(* IEC 61131-3 sources: myCodes/Stone/07.02.2022 - OOPs Approach/MPx_One_New/Mpx_One_Source_Code/MPx_One/3. USHPXMPX010A1/USHPXMPX010A1/MPXone_Medium/Gui/Actions, 31 files *)

(* ---- ALM_HystPROGRAM_RELEASE.st ---- *)
USING System;
USING System.UI;
USING HEOneRow;

FUNCTION ALM_HystPROGRAM_RELEASE
	VAR_INPUT
		keyPressed:UINT;
		keyCounter:UINT;
	END_VAR

    currMenuLevel := 2;

    GoToLoop(LoopList#ALM_LOG);

END_FUNCTION

(* ---- ALM_menu_ESC_PROGRAM_RELEASE.st ---- *)
USING System;
USING System.UI;
USING HEOneRow;

FUNCTION ALM_menu_ESC_PROGRAM_RELEASE
	VAR_INPUT
		keyPressed:UINT;
		keyCounter:UINT;
	END_VAR

    currMenuLevel := 1;
    currMenu := 4;
    GoToMask(MaskList#ALM);

END_FUNCTION

(* ---- ALM_ParamPROGRAM_RELEASE.st ---- *)
USING System;
USING System.UI;
USING HEOneRow;

FUNCTION ALM_ParamPROGRAM_RELEASE
	VAR_INPUT
		keyPressed:UINT;
		keyCounter:UINT;
	END_VAR

    currMenuLevel := 2;
    GoToLoop(LoopList#ALM_Param);

END_FUNCTION

(* ---- checkPassword.st ---- *)
USING System;
USING System.UI;
USING HEOneRow;

FUNCTION checkPassword
	VAR_INPUT
		keyPressed:UINT;
		keyCounter:UINT;
	END_VAR

    IF tmpPassword = TO_USINT(PwdDisplay) THEN
        GoToLoop(LoopList#Menu);
        blockHmi := TRUE;

        tmpPassword := 0;

        currMenu := 1; // Vis Menu
        currMenuLevel := 0; // Menu level
    ELSE
        // Wrong password
        LedBlinkArrow := FALSE;
        WrongPsw := TRUE;
        blockHmi := TRUE;
        GoToLoop(LoopList#Main);
    END_IF;

END_FUNCTION

(* ---- CntPRG.st ---- *)
USING System;
USING System.UI;
USING HEOneRow;

FUNCTION CntPRG
	VAR_INPUT
		keyPressed:UINT;
		keyCounter:UINT;
	END_VAR

    //DispMngInst.StartSync(DownloadDir#ACUtoHMI);
    NewDispPrompt := FALSE;
    GoToLoop(LoopList#Main);

END_FUNCTION

(* ---- Dir_CleanPRG.st ---- *)
USING System;
USING System.UI;
USING HEOneRow;

FUNCTION Dir_CleanPRG
	VAR_INPUT
		keyPressed:UINT;
		keyCounter:UINT;
	END_VAR

    ManClean := NOT ManClean;
END_FUNCTION

(* ---- Dir_ContCyclPRG.st ---- *)
USING System;
USING System.UI;
USING HEOneRow;

FUNCTION Dir_ContCyclPRG
	VAR_INPUT
		keyPressed:UINT;
		keyCounter:UINT;
	END_VAR

    ManContCycle_byDisplay := NOT ManContCycle_byDisplay;

END_FUNCTION

(* ---- Dir_DefrostPRG.st ---- *)
USING System;
USING System.UI;
USING HEOneRow;

FUNCTION Dir_DefrostPRG
	VAR_INPUT
		keyPressed:UINT;
		keyCounter:UINT;
	END_VAR

    ManDfr := NOT ManDfr;

END_FUNCTION

(* ---- Dir_LightPRG.st ---- *)
USING System;
USING System.UI;
USING HEOneRow;

FUNCTION Dir_LightPRG
	VAR_INPUT
		keyPressed:UINT;
		keyCounter:UINT;
	END_VAR

    LightsOn := NOT LightsOn;
END_FUNCTION

(* ---- Dir_NetDefrostPRG.st ---- *)
USING System;
USING System.UI;
USING HEOneRow;

FUNCTION Dir_NetDefrostPRG
	VAR_INPUT
		keyPressed:UINT;
		keyCounter:UINT;
	END_VAR

    NetworkDfr := NOT NetworkDfr;

END_FUNCTION

(* ---- Dir_OnOffPRG.st ---- *)
USING System;
USING System.UI;
USING HEOneRow;

FUNCTION Dir_OnOffPRG
	VAR_INPUT
		keyPressed:UINT;
		keyCounter:UINT;
	END_VAR

    IF NOT(DigitalInputs.Fct.RemoteOff) THEN // TRAC #99: Allow to change the status from UI only if remote off is not active
        KeyboardOnOff := NOT KeyboardOnOff;
        //        UnitStatus := NOT UnitStatus;
    END_IF;

END_FUNCTION

(* ---- DisPRG.st ---- *)
USING System;
USING System.UI;
USING HEOneRow;

FUNCTION DisPRG
	VAR_INPUT
		keyPressed:UINT;
		keyCounter:UINT;
	END_VAR

    //DispMngInst.StartSync(DownloadDir#HMItoACU);
    NewDispPrompt := FALSE;
    GoToLoop(LoopList#Main);

END_FUNCTION

(* ---- doNothing.st ---- *)
USING System;
USING System.UI;
USING HEOneRow;

FUNCTION doNothing
	VAR_INPUT
		keyPressed:UINT;
		keyCounter:UINT;
	END_VAR

END_FUNCTION

(* ---- GlassGUIALARM.st ---- *)
USING System;
USING System.UI;
USING HEOneRow;

FUNCTION GlassGUIALARM
	VAR_INPUT
		keyPressed:UINT;
		keyCounter:UINT;
	END_VAR

    IF AckAlm AND keyCounter < 30 THEN
        // Block user interface
        IF NOT EnKeyboard THEN
            RETURN;
        END_IF;

        IF (NOT OrAlrm) AND (NOT OrWarning) THEN
            RETURN;
        END_IF;

        GoToMask(MaskList#ActiveAlarms);
        //InsideLoopAlrm := TRUE;
        Navigation := TRUE;
    END_IF;

    IF NOT Alarms.Al.Warn_Door.Info.Trigger THEN
        AckAlm := TRUE;
    END_IF;

END_FUNCTION

(* ---- GoToLastRTC.st ---- *)
USING System;
USING System.UI;
USING HEOneRow;

FUNCTION GoToLastRTC
	VAR_INPUT
		keyPressed:UINT;
		keyCounter:UINT;
	END_VAR

    //GoToMask(MaskList#tc);
END_FUNCTION

(* ---- GoToMain.st ---- *)
USING System;
USING System.UI;
USING HEOneRow;

FUNCTION GoToMain
	VAR_INPUT
		keyPressed:UINT;
		keyCounter:UINT;
	END_VAR

    // Turn off LEDS used for menu
    LedOnArrow := FALSE;
    LedBlinkArrow := FALSE;

    /*rkLed[0] := FALSE;
    rkLed[1] := FALSE;
    rkLed[2] := FALSE;
    rkLed[3] := FALSE;
    lkLed[0] := FALSE;
    lkLed[1] := FALSE;
    lkLed[2] := FALSE;
    lkLed[3] := FALSE;
    lkLed[4] := FALSE;
    LedAlarm := FALSE;*/

    Navigation := FALSE;
    InsideLoopDirFunct := FALSE;
    currMenuLevel := 0;

    blockHmi := TRUE;
    BasicVisualiz := FALSE;

    GoToMask(MaskList#mMain);
END_FUNCTION

(* ---- GoToPassword.st ---- *)
USING System;
USING System.UI;
USING HEOneRow;

FUNCTION GoToPassword
	VAR_INPUT
		keyPressed:UINT;
		keyCounter:UINT;
	END_VAR

    // Block user interface
    IF NOT EnKeyboard THEN
        RETURN;
    END_IF;

    IF keyCounter>30 AND BlockHmi = FALSE THEN
        blockHmi := TRUE;
        Navigation := TRUE;
        GoToMask(MaskList#mPassword);
    END_IF;

END_FUNCTION

(* ---- HSx_PROGRAM_RELEASE.st ---- *)
USING System;
USING System.UI;
USING HEOneRow;

FUNCTION HSx_PROGRAM_RELEASE
	VAR_INPUT
		keyPressed:UINT;
		keyCounter:UINT;
	END_VAR

    CASE GetCurrentMask() OF
        TO_UINT(MaskList#HS0) : IdxVis_AlrmHyst := 1;
        TO_UINT(MaskList#HS1) : IdxVis_AlrmHyst := 2;
        TO_UINT(MaskList#HS2) : IdxVis_AlrmHyst := 3;
        TO_UINT(MaskList#HS3) : IdxVis_AlrmHyst := 4;
        TO_UINT(MaskList#HS4) : IdxVis_AlrmHyst := 5;
        TO_UINT(MaskList#HS5) : IdxVis_AlrmHyst := 6;
        TO_UINT(MaskList#HS6) : IdxVis_AlrmHyst := 7;
        TO_UINT(MaskList#HS7) : IdxVis_AlrmHyst := 8;
        TO_UINT(MaskList#HS8) : IdxVis_AlrmHyst := 9;
        TO_UINT(MaskList#HS9) : IdxVis_AlrmHyst := 10;
    END_CASE;

   GoToMask(MaskList#ShowAlrmHyst);

END_FUNCTION

(* ---- MenuPRG.st ---- *)
USING System;
USING System.UI;
USING HEOneRow;

FUNCTION MenuPRG
	VAR_INPUT
		keyPressed:UINT;
		keyCounter:UINT;
	END_VAR

    IF keyCounter >30 AND NOT blockHmi THEN
        blockHmi := TRUE;

        IF currMenuLevel = 0 THEN
            GoToMask(MaskList#mMain);

        ELSE
            CASE currMenu OF
                1: GoToMask(MaskList#VIS);
                2: GoToMask(MaskList#CTL);
                3: GoToMask(MaskList#DEF);
                4: GoToMask(MaskList#ALM);
                5: GoToMask(MaskList#FAN);
                6: GoToMask(MaskList#EVD);
                7: GoToMask(MaskList#CNF);
            ELSE
                GoToLoop(LoopList#Menu);
            END_CASE;

            currMenuLevel := 0;
        END_IF;
    END_IF;

END_FUNCTION

(* ---- MenuPROGRAM_RELEASE.st ---- *)
USING System;
USING System.UI;

NAMESPACE HEOneRow

FUNCTION MenuPROGRAM_RELEASE
	VAR_INPUT
		keyPressed:UINT;
		keyCounter:UINT;
	END_VAR

    IF keyCounter < 30 AND NOT blockHmi THEN

        IF BasicVisualiz AND GetCurrentMask() = GetLastMaskInLoop(gui.currentLoop) THEN
            GoToMask(MaskList#mMain);
            BasicVisualiz := FALSE;
            LedOnArrow := FALSE;
            PrbVisualiz := FALSE;
            RETURN;
        END_IF;

        CASE currMenuLevel OF
            0: // At function selection

            IF isProdBasicVersion AND currMenu = 6 THEN
                currMenu := 7;
            END_IF;

            CASE currMenu OF
                1: GoToLoop(LoopList#VIS_Loop);
                2: GoToLoop(LoopList#CTL_Param);
                3: GoToLoop(LoopList#dEF_Param);
                4: GoToLoop(LoopList#ALM_menu);
                5: GoToLoop(LoopList#FAN_Param);
                {IF DEF(MPXONE_MEDIUM)}
                6: GoToLoop(LoopList#EVD_Param);
                {ENDIF}
                7: GoToLoop(LoopList#CNF_Param);
                8: GoToLoop(LoopList#rtC_Param);
            ELSE
                GoToLoop(LoopList#Menu);
            END_CASE;

            currMenuLevel := 1;

            1: // editing the value
            GoToNextField();

            // Or exiting
            IF GetCurrentMask() = GetLastMaskInLoop(gui.currentLoop) THEN
                CASE currMenu OF
                    1: GoToMask(MaskList#VIS);
                    2: GoToMask(MaskList#CTL);
                    3: GoToMask(MaskList#DEF);
                    4: GoToMask(MaskList#ALM);
                    5: GoToMask(MaskList#FAN);
                    6: GoToMask(MaskList#EVD);
                    7: GoToMask(MaskList#CNF);
                    8: GoToMask(MaskList#RtC);
                ELSE
                    GoToLoop(LoopList#Menu);
                END_CASE;

                currMenuLevel := 0;
                currMenu_SecondLev := 0;
            END_IF;

            2: // editing the value
            GoToNextField();

            // Or exiting
            IF GetCurrentMask() = GetLastMaskInLoop(gui.currentLoop) THEN
                CASE currMenu_SecondLev OF
                    0: GoToMask(MaskList#ALM_Param);
                    1: GoToMask(MaskList#ALM_Hyst);
                ELSE
                    GoToMask(MaskList#ALM);
                END_CASE;
                currMenu := 4;
                currMenuLevel := 1;
            END_IF;

        END_CASE;

    END_IF;

    blockHmi := FALSE;

END_FUNCTION

END_NAMESPACE

(* ---- MenuSecondUPDOWN.st ---- *)
USING System;
USING System.UI;
USING HEOneRow;

FUNCTION MenuSecondUPDOWN
	VAR_INPUT
		keyPressed:UINT;
		keyCounter:UINT;
	END_VAR

    // keyPressed = 14 tasto UP
    IF keyPressed = 14 THEN
        currMenu_SecondLev := currMenu_SecondLev - 1;
        IF currMenu_SecondLev > 2 THEN // CurrMenu is unsigned so it will become 255 insthead of -1
            currMenu_SecondLev := 2;
        END_IF;
        GoToPreviousMask();
    END_IF;

    // keyPressed = 15 tasto DOWN
    IF keyPressed = 15 THEN
        currMenu_SecondLev := currMenu_SecondLev + 1;
        IF currMenu_SecondLev > 2 THEN
            currMenu_SecondLev := 0;
        END_IF;
        GoToNextMask();
    END_IF;

END_FUNCTION

(* ---- MenuUPDOWN.st ---- *)
USING System;
USING System.UI;
USING HEOneRow;

FUNCTION MenuUPDOWN
	VAR_INPUT
		keyPressed:UINT;
		keyCounter:UINT;
	END_VAR

    // keyPressed = 14 tasto UP
    IF keyPressed = 14 THEN
        currMenu := currMenu - 1;
        IF currMenu > MENU_ITEMS THEN // CurrMenu is unsigned so it will become 255 insthead of -1
            currMenu := MENU_ITEMS;
        END_IF;
        GoToPreviousMask();
    END_IF;

    // keyPressed = 15 tasto DOWN
    IF keyPressed = 15 THEN
        currMenu := currMenu + 1;
        IF currMenu > MENU_ITEMS THEN
            currMenu := 0;
        END_IF;
        GoToNextMask();
    END_IF;

END_FUNCTION

(* ---- mMainALARM.st ---- *)
USING System;
USING System.UI;
USING HEOneRow;

FUNCTION mMainALARM
	VAR_INPUT
		keyPressed:UINT;
		keyCounter:UINT;
	END_VAR

//    IF AckAlm THEN
//        GoToMask(MaskList#ActiveAlarms);
//        //InsideLoopAlrm := TRUE;
//        Navigation := TRUE;
//    END_IF;

    // Block user interface
    IF NOT EnKeyboard THEN
        RETURN;
    END_IF;

    // Long press to reset alarm
    IF keyCounter>30 AND blockHmi = FALSE THEN
        AlrmRes := TRUE;
    END_IF;

END_FUNCTION

(* ---- mMainPRG.st ---- *)
USING System;
USING System.UI;
USING HEOneRow;

FUNCTION mMainPRG
	VAR_INPUT
		keyPressed:UINT;
		keyCounter:UINT;
	END_VAR

    IF keyCounter>30 AND firstCycle AND NOT blockHmi THEN
        blockHmi := TRUE;
        StartupReset := TRUE;
        GoToMask(MaskList#DefSelection);
        RETURN;
    END_IF;

    IF firstCycle THEN
        RETURN;
    END_IF;

    // Block user interface
    IF NOT EnKeyboard THEN
        RETURN;
    END_IF;

    IF keyCounter>30 AND blockHmi = FALSE THEN
        blockHmi := TRUE;
        Navigation := TRUE;
        GoToMask(MaskList#mTxtPsd);
    END_IF;

END_FUNCTION

(* ---- mMainPROGRAM_RELEASE.st ---- *)
USING System;
USING System.UI;
USING HEOneRow;

FUNCTION mMainPROGRAM_RELEASE
	VAR_INPUT
		keyPressed:UINT;
		keyCounter:UINT;
	END_VAR

    // Block user interface
    IF NOT EnKeyboard THEN
        RETURN;
    END_IF;

    Navigation := FALSE;
    InsideLoopDirFunct := FALSE;

    IF blockHmi = FALSE AND keyCounter <30 AND EnDirFunct AND NOT firstCycle THEN
        Navigation := TRUE;
        InsideLoopDirFunct := TRUE;
        LedBlinkArrow := FALSE;
        LedOnArrow := TRUE;
        blockHmi := TRUE;

        GoToLoop(LoopList#DirFunction);
    END_IF;

    blockHmi := FALSE;

END_FUNCTION

(* ---- mMainUPDOWN.st ---- *)
USING System;
USING System.UI;
USING HEOneRow;

FUNCTION mMainUPDOWN
	VAR_INPUT
		keyPressed:UINT;
		keyCounter:UINT;
	END_VAR

    // Block user interface
    IF NOT EnKeyboard THEN
        RETURN;
    END_IF;

    Navigation := TRUE;
    BasicVisualiz := TRUE;
    PrbVisualiz := TRUE;
    LedOnArrow := TRUE;
    currMenuLevel := 1;

    GoToLoop(LoopList#VIS_Loop);

END_FUNCTION

(* ---- mTxtPsdPRG.st ---- *)
USING System;
USING System.UI;
USING HEOneRow;

FUNCTION mTxtPsdPRG
	VAR_INPUT
		keyPressed:UINT;
		keyCounter:UINT;
	END_VAR

    IF NOT blockHmi THEN
        LedOnArrow := FALSE;
        LedBlinkArrow := TRUE;
        GoToMask(MaskList#mPassword);
    END_IF;

END_FUNCTION

(* ---- mTxtPsdPROGRAM_RELEASE.st ---- *)
USING System;
USING System.UI;
USING HEOneRow;

FUNCTION mTxtPsdPROGRAM_RELEASE
	VAR_INPUT
		keyPressed:UINT;
		keyCounter:UINT;
	END_VAR

    blockHmi := FALSE;

END_FUNCTION

(* ---- PasswordDOWN.st ---- *)
USING System;
USING System.UI;
USING HEOneRow;

FUNCTION PasswordDOWN
	VAR_INPUT
		keyPressed:UINT;
		keyCounter:UINT;
	END_VAR

   tmpPassword := tmpPassword - 1;
END_FUNCTION

(* ---- PasswordUP.st ---- *)
USING System;
USING System.UI;
USING HEOneRow;

FUNCTION PasswordUP
	VAR_INPUT
		keyPressed:UINT;
		keyCounter:UINT;
	END_VAR

    tmpPassword := tmpPassword + 1;
END_FUNCTION

(* ---- WIZ_ENDPRG.st ---- *)
USING System;
USING System.UI;
USING HEOneRow;

FUNCTION WIZ_ENDPRG
	VAR_INPUT
		keyPressed:UINT;
		keyCounter:UINT;
	END_VAR

    // Configure the probes
    Ain_Types.Group1 := tmpWiz.Fct._P1.usint;
    Ain_Types.Group2 := tmpWiz.Fct._P2.usint;
    Ain_Types.Group3 := tmpWiz.Fct._P3.usint;

    Ain_Cfg.Fct.SuctT.Ch := TO_SINT(tmpWiz.Fct._FD.usint);
    Ain_Cfg.Fct.EvapP.Ch := TO_SINT(tmpWiz.Fct._FE.usint);

    // Probe limits
    EvapMax := tmpWiz.Fct._UE.real;
    EvapMin := tmpWiz.Fct._LE.real;

    // Valve configuration
    ValveCnf := tmpWiz.Fct.P1.usint;
    RfrgTyp := TO_UINT(tmpWiz.Fct.PH.usint);

    // Configure protocols
    BMS_Addr := tmpWiz.Fct.H0.usint;
    BMS_Prot := tmpWiz.Fct.H3.bool;
    isMaster := tmpWiz.Fct.In.bool;
    SlavesNum := tmpWiz.Fct.Sn.usint;

    // Wizard flags to complete the procedure
    WizDone := TRUE;
    WizProgress := FALSE;
    blockHmi := TRUE;
    StartupReset := FALSE;

    // Force backup
    //RetainForceBackup();
    GoToLoop(LoopList#Main);
    //SoftwareReset(ResetMode#Warm);

    LedOnArrow := FALSE;

END_FUNCTION
